Omron CX-Programmer project NewProject (CX-Programmer 9.75)

# PLC NewPLC1: CJ2M CPU11

## Global symbols (name address type ; comment)
LAMPU1 FunctionBlock1

## Program NewProgram1 (cyclic task 0)
Local symbols
LAMPU 100.00 BOOL
START 0.00 BOOL
STOP 0.01 BOOL

### Section Section1

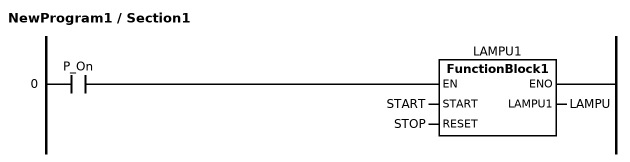
; rung 0
LD P_On
CALL LAMPU1 : FunctionBlock1 (START := START, RESET := STOP, LAMPU1 => LAMPU)

### Section END
; rung 0
END(001)

## Function block FunctionBlock1
VAR_INPUT
  START : BOOL;
  RESET : BOOL;
  SENSOR_5cm : BOOL;
END_VAR
VAR_OUTPUT
  LAMPU1 : BOOL;
  CONVEYOR : BOOL;
  indikator5cm : BOOL;
END_VAR
VAR
  MULAI : BOOL;
  TIMER : TIMER;
  COUNTER1 : COUNTER;
END_VAR

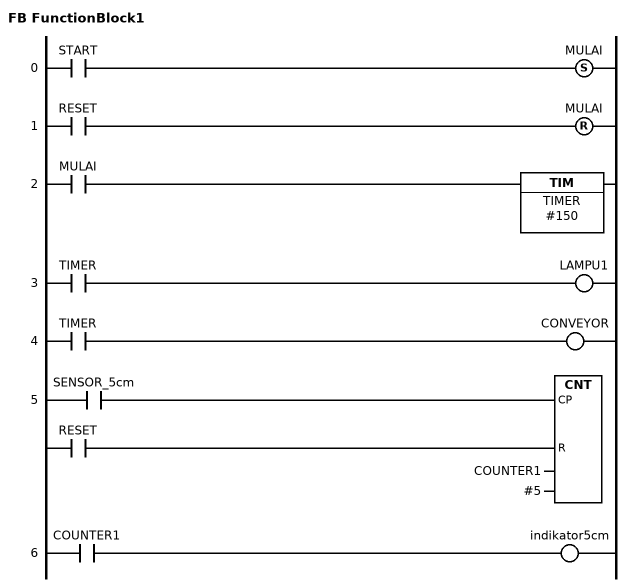
; rung 0
LD START
SET MULAI
; rung 1
LD RESET
RSET MULAI
; rung 2
LD MULAI
TIM TIMER #150
; rung 3
LD TIMER
OUT LAMPU1
; rung 4
LD TIMER
OUT CONVEYOR
; rung 5
LD SENSOR_5cm
LD RESET
CNT COUNTER1 #5
; rung 6
LD COUNTER1
OUT indikator5cm